// TIA Portal project "Lab2_V18" (V18)

(* hardware
DEVICE "S7300/ET200M station_1"  S7-300 station
   slot 0: "Rail_0"  Rail  6ES7 390-1***0-0AA0
   slot 2: "PLC_1"  CPU 314C-2 DP  6ES7 314-6CG03-0AB0  V2.6
      slot 0: "MPI interface_1"  X1
      slot 1: "DP interface_1"  X2
      slot 2: "DI 24/DO 16_1"  DI24/DO16
      slot 3: "AI 5/AO 2_1"  AI5/AO2
      slot 4: "Count_1"  Counter
      slot 5: "Positioning_1"  Positioning
   slot 4: "CP 340 RS232C_1"  CP 340 RS232C  6ES7 340-1AH02-0AE0  V1.0
DEVICE "S7-300/ET200M station_1"  S7-300 station
   slot 0: "Rail_0"  Rail  6ES7 390-1***0-0AA0
   slot 2: "PLC_2"  CPU 314C-2 DP  6ES7 314-6CG03-0AB0  V2.6
      slot 0: "MPI interface_1"  X1
      slot 1: "DP interface_1"  X2
      slot 2: "DI 24/DO 16_1"  DI24/DO16
      slot 3: "AI 5/AO 2_1"  AI5/AO2
      slot 4: "Count_1"  Counter
      slot 5: "Positioning_1"  Positioning
*)

// ===== PLC "PLC_1"  CPU 314C-2 DP =====

VAR_GLOBAL   // PLC tag table "Default tag table"
   "step0" AT %M0.0 : Bool;
   "step1" AT %M0.1 : Bool;
   "step2" AT %M0.2 : Bool;
   "step3" AT %M0.3 : Bool;
   "step4" AT %M0.4 : Bool;
   "step5" AT %M0.5 : Bool;
   "step6" AT %M0.6 : Bool;
   "step7" AT %M0.7 : Bool;
   "step8" AT %M1.0 : Bool;
   "timer1" AT %M1.1 : Bool;
   "timer2" AT %M1.2 : Bool;
   "FS" AT %M1.3 : Bool;
   "startbutton" AT %I125.0 : Bool;
END_VAR

VAR_GLOBAL   // PLC tag table "Tag table_1"
   "sp1e" AT %I124.6 : Bool;
   "sp1r" AT %I124.7 : Bool;
   "sp2e" AT %I124.5 : Bool;
   "sp2r" AT %I124.4 : Bool;
   "GR" AT %Q124.7 : Bool;
   "cmdP1e" AT %Q124.5 : Bool;
   "cmdP1r" AT %Q124.6 : Bool;
   "cmdP2e" AT %Q124.3 : Bool;
   "cmdP2r" AT %Q124.4 : Bool;
END_VAR

FUNCTION "Block_1" : Void   // FC1, STL
{ S7_Optimized_Access := 'FALSE' }
VERSION : 0.1
BEGIN

REGION Network 1
         A     "step0";
         AN    "step1";

         O(;
         A     "step8";
         A     "sp1r";
         );
         O(;

         A     "FS";


         );

         =     "step0";

         R     "FS";
END_REGION

REGION Network 2
         A     "step0";
         A     "startbutton";
         O(;
         A     "step1";
         AN    "step2";

         );


         =     "step1";
END_REGION

REGION Network 3
   //(
         A     "sp2e";


         A     "step1";
         O(;
         A     "step2";
         AN    "step3";

         );
   //      )
         =     "step2";
END_REGION

REGION Network 4
         A     "step2";
         A     "timer1";
         O(;
         A     "step3";
         AN    "step4";

         );
         =     "step3";
END_REGION

REGION Network 5
         A     "step3";
         A     "sp2r";
         O(;
         A     "step4";
         AN    "step5";

         );
         =     "step4";
END_REGION

REGION Network 6
         A     "step4";
         A     "sp1e";
         O(;
         A     "step5";
         AN    "step6";

         );
         =     "step5";
END_REGION

REGION Network 7
         A     "step5";
         A     "sp2r";
         O(;
         A     "step6";
         AN    "step7";

         );
         =     "step6";
END_REGION

REGION Network 8
         A     "step6";

         A     "timer2";
         O(;
         A     "step7";

         AN    "step8";


         );
         =     "step7";
END_REGION

REGION Network 9
         A     "step7";

         A     "sp2r";
         O(;
         A     "step8";
         AN    "step0";

         );
         =     "step8";
END_REGION

REGION Network 10
         A     "step4";
         =     "cmdP1e";
END_REGION

REGION Network 11
         A     "step8";
         =     "cmdP1r";
END_REGION

REGION Network 12
         A     "step1";
         O     "step5";
         =     "cmdP2e";
END_REGION

REGION Network 13
         A     "step3";
         O     "step7";
         =     "cmdP2r";
END_REGION

REGION Network 14
         A     "step2";
         O     "step3";
         O     "step4";
         O     "step5";
         =     "GR";
END_REGION

REGION Network 15
         A     "step2";
         A     "IEC_Timer_0_DB".IN;
         =     "timer1";
END_REGION

REGION Network 16
         A     "step6";
         A     "IEC_Timer_0_DB".IN;
         =     "timer2";
END_REGION
END_FUNCTION

FUNCTION "Block_2" : Void   // FC2, LAD
{ S7_Optimized_Access := 'FALSE' }
VERSION : 0.1
BEGIN

REGION Network 2
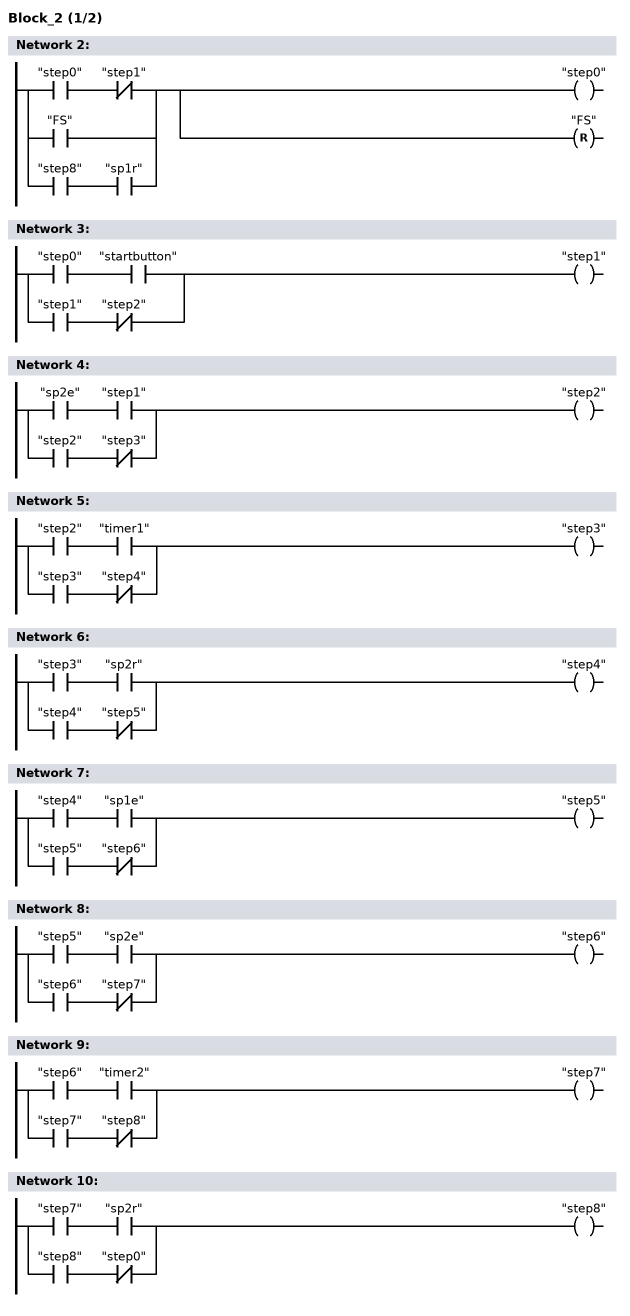
   RUNG wire#powerrail
      Contact( "step0" )
      I_Contact( "step1" )
      wire#w1
      Coil( "step0" )
   END_RUNG
   RUNG wire#powerrail
      Contact( "FS" )
   END_RUNG wire#w1
   RUNG wire#powerrail
      Contact( "step8" )
      Contact( "sp1r" )
   END_RUNG wire#w1
   RUNG wire#w1
      R_Coil( "FS" )
   END_RUNG
   // the same network as SCL:
   "step0" := ("step0" AND NOT "step1") OR "FS" OR ("step8" AND "sp1r");
   IF "step0" THEN "FS" := FALSE; END_IF;
END_REGION

REGION Network 3
   RUNG wire#powerrail
      Contact( "step0" )
      Contact( "startbutton" )
      wire#w1
      Coil( "step1" )
   END_RUNG
   RUNG wire#powerrail
      Contact( "step1" )
      I_Contact( "step2" )
   END_RUNG wire#w1
   // the same network as SCL:
   "step1" := ("step0" AND "startbutton") OR ("step1" AND NOT "step2");
END_REGION

REGION Network 4
   RUNG wire#powerrail
      Contact( "sp2e" )
      Contact( "step1" )
      wire#w1
      Coil( "step2" )
   END_RUNG
   RUNG wire#powerrail
      Contact( "step2" )
      I_Contact( "step3" )
   END_RUNG wire#w1
   // the same network as SCL:
   "step2" := ("sp2e" AND "step1") OR ("step2" AND NOT "step3");
END_REGION

REGION Network 5
   RUNG wire#powerrail
      Contact( "step2" )
      Contact( "timer1" )
      wire#w1
      Coil( "step3" )
   END_RUNG
   RUNG wire#powerrail
      Contact( "step3" )
      I_Contact( "step4" )
   END_RUNG wire#w1
   // the same network as SCL:
   "step3" := ("step2" AND "timer1") OR ("step3" AND NOT "step4");
END_REGION

REGION Network 6
   RUNG wire#powerrail
      Contact( "step3" )
      Contact( "sp2r" )
      wire#w1
      Coil( "step4" )
   END_RUNG
   RUNG wire#powerrail
      Contact( "step4" )
      I_Contact( "step5" )
   END_RUNG wire#w1
   // the same network as SCL:
   "step4" := ("step3" AND "sp2r") OR ("step4" AND NOT "step5");
END_REGION

REGION Network 7
   RUNG wire#powerrail
      Contact( "step4" )
      Contact( "sp1e" )
      wire#w1
      Coil( "step5" )
   END_RUNG
   RUNG wire#powerrail
      Contact( "step5" )
      I_Contact( "step6" )
   END_RUNG wire#w1
   // the same network as SCL:
   "step5" := ("step4" AND "sp1e") OR ("step5" AND NOT "step6");
END_REGION

REGION Network 8
   RUNG wire#powerrail
      Contact( "step5" )
      Contact( "sp2e" )
      wire#w1
      Coil( "step6" )
   END_RUNG
   RUNG wire#powerrail
      Contact( "step6" )
      I_Contact( "step7" )
   END_RUNG wire#w1
   // the same network as SCL:
   "step6" := ("step5" AND "sp2e") OR ("step6" AND NOT "step7");
END_REGION

REGION Network 9
   RUNG wire#powerrail
      Contact( "step6" )
      Contact( "timer2" )
      wire#w1
      Coil( "step7" )
   END_RUNG
   RUNG wire#powerrail
      Contact( "step7" )
      I_Contact( "step8" )
   END_RUNG wire#w1
   // the same network as SCL:
   "step7" := ("step6" AND "timer2") OR ("step7" AND NOT "step8");
END_REGION

REGION Network 10
   RUNG wire#powerrail
      Contact( "step7" )
      Contact( "sp2r" )
      wire#w1
      Coil( "step8" )
   END_RUNG
   RUNG wire#powerrail
      Contact( "step8" )
      I_Contact( "step0" )
   END_RUNG wire#w1
   // the same network as SCL:
   "step8" := ("step7" AND "sp2r") OR ("step8" AND NOT "step0");
END_REGION

REGION Network 11
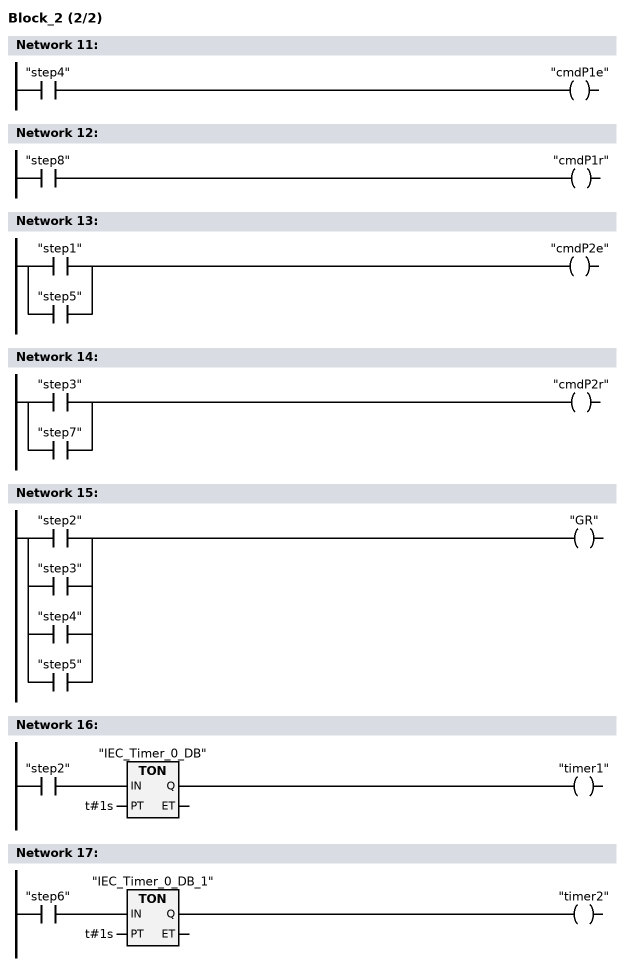
   RUNG wire#powerrail
      Contact( "step4" )
      Coil( "cmdP1e" )
   END_RUNG
   // the same network as SCL:
   "cmdP1e" := "step4";
END_REGION

REGION Network 12
   RUNG wire#powerrail
      Contact( "step8" )
      Coil( "cmdP1r" )
   END_RUNG
   // the same network as SCL:
   "cmdP1r" := "step8";
END_REGION

REGION Network 13
   RUNG wire#powerrail
      Contact( "step1" )
      wire#w1
      Coil( "cmdP2e" )
   END_RUNG
   RUNG wire#powerrail
      Contact( "step5" )
   END_RUNG wire#w1
   // the same network as SCL:
   "cmdP2e" := "step1" OR "step5";
END_REGION

REGION Network 14
   RUNG wire#powerrail
      Contact( "step3" )
      wire#w1
      Coil( "cmdP2r" )
   END_RUNG
   RUNG wire#powerrail
      Contact( "step7" )
   END_RUNG wire#w1
   // the same network as SCL:
   "cmdP2r" := "step3" OR "step7";
END_REGION

REGION Network 15
   RUNG wire#powerrail
      Contact( "step2" )
      wire#w1
      Coil( "GR" )
   END_RUNG
   RUNG wire#powerrail
      Contact( "step3" )
   END_RUNG wire#w1
   RUNG wire#powerrail
      Contact( "step4" )
   END_RUNG wire#w1
   RUNG wire#powerrail
      Contact( "step5" )
   END_RUNG wire#w1
   // the same network as SCL:
   "GR" := "step2" OR "step3" OR "step4" OR "step5";
END_REGION

REGION Network 16
   "IEC_Timer_0_DB".TON(IN := "step2", PT := t#1s);
   "timer1" := "IEC_Timer_0_DB".Q;
END_REGION

REGION Network 17
   "IEC_Timer_0_DB_1".TON(IN := "step6", PT := t#1s);
   "timer2" := "IEC_Timer_0_DB_1".Q;
END_REGION
END_FUNCTION

FUNCTION "Block_3" : Void   // FC3, SCL
{ S7_Optimized_Access := 'FALSE' }
VERSION : 0.1
BEGIN
   "step0" := ("step0" AND NOT "step1")
   OR ("step8" AND "sp1r")
   OR "FS";
   IF "step0"  THEN
       "FS" := FALSE;
       // Statement section IF
      ;
   END_IF;

   "IEC_Timer_0_DB_2".TON(IN:="step2",
                          PT:=t#1s,
                          Q=>"timer1");
END_FUNCTION

ORGANIZATION_BLOCK "Main"   // OB1, LAD
TITLE = "Main Program Sweep (Cycle)"
{ S7_Optimized_Access := 'FALSE' }
VERSION : 0.1
   VAR_TEMP
      OB1_EV_CLASS : Byte;   // Bits 0-3 = 1 (Coming event), Bits 4-7 = 1 (Event class 1)
      OB1_SCAN_1 : Byte;   // 1 (Cold restart scan 1 of OB 1), 3 (Scan 2-n of OB 1)
      OB1_PRIORITY : Byte;   // Priority of OB Execution
      OB1_OB_NUMBR : Byte;   // 1 (Organization block 1, OB1)
      OB1_RESERVED_1 : Byte;   // Reserved for system
      OB1_RESERVED_2 : Byte;   // Reserved for system
      OB1_PREV_CYCLE : Int;   // Cycle time of previous OB1 scan (milliseconds)
      OB1_MIN_CYCLE : Int;   // Minimum cycle time of OB1 (milliseconds)
      OB1_MAX_CYCLE : Int;   // Maximum cycle time of OB1 (milliseconds)
      OB1_DATE_TIME : Date_And_Time;   // Date and time OB1 started
   END_VAR
BEGIN

REGION Network 1
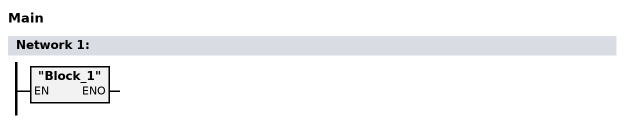
   RUNG wire#powerrail
      "Block_1"()
   END_RUNG
   // the same network as SCL:
   "Block_1"();
END_REGION
END_ORGANIZATION_BLOCK

ORGANIZATION_BLOCK "COMPLETE RESTART"   // OB100, LAD
TITLE = "Complete Restart"
{ S7_Optimized_Access := 'FALSE' }
VERSION : 0.1
   VAR_TEMP
      OB100_EV_CLASS : Byte;   // 16#13, Event class 1, Entering event state, Event logged in diagnostic buffer
      OB100_STRTUP : Byte;   // 16#81/82/83/84 Method of startup
      OB100_PRIORITY : Byte;   // Priority of OB Execution
      OB100_OB_NUMBR : Byte;   // 100 (Organization block 100, OB100)
      OB100_RESERVED_1 : Byte;   // Reserved for system
      OB100_RESERVED_2 : Byte;   // Reserved for system
      OB100_STOP : Word;   // Event that caused CPU to stop (16#4xxx)
      OB100_STRT_INFO : DWord;   // Information on how system started
      OB100_DATE_TIME : Date_And_Time;   // Date and time OB100 started
   END_VAR
BEGIN

REGION Network 1
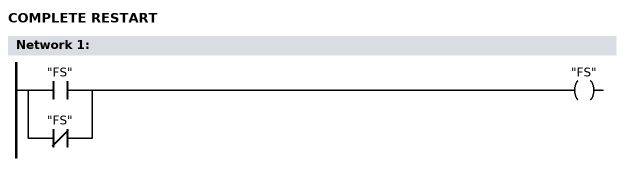
   RUNG wire#powerrail
      Contact( "FS" )
      wire#w1
      Coil( "FS" )
   END_RUNG
   RUNG wire#powerrail
      I_Contact( "FS" )
   END_RUNG wire#w1
   // the same network as SCL:
   "FS" := "FS" OR NOT "FS";
END_REGION
END_ORGANIZATION_BLOCK

// ===== PLC "PLC_2"  CPU 314C-2 DP =====

ORGANIZATION_BLOCK "Main"   // OB1, LAD
TITLE = "Main Program Sweep (Cycle)"
{ S7_Optimized_Access := 'FALSE' }
VERSION : 0.1
   VAR_TEMP
      OB1_EV_CLASS : Byte;   // Bits 0-3 = 1 (Coming event), Bits 4-7 = 1 (Event class 1)
      OB1_SCAN_1 : Byte;   // 1 (Cold restart scan 1 of OB 1), 3 (Scan 2-n of OB 1)
      OB1_PRIORITY : Byte;   // Priority of OB Execution
      OB1_OB_NUMBR : Byte;   // 1 (Organization block 1, OB1)
      OB1_RESERVED_1 : Byte;   // Reserved for system
      OB1_RESERVED_2 : Byte;   // Reserved for system
      OB1_PREV_CYCLE : Int;   // Cycle time of previous OB1 scan (milliseconds)
      OB1_MIN_CYCLE : Int;   // Minimum cycle time of OB1 (milliseconds)
      OB1_MAX_CYCLE : Int;   // Maximum cycle time of OB1 (milliseconds)
      OB1_DATE_TIME : Date_And_Time;   // Date and time OB1 started
   END_VAR
BEGIN
END_ORGANIZATION_BLOCK